TYPE ST_LA_Stellwert :
STRUCT

	Aussenluftklappe_Stellung 		: REAL;
	Bypassklappe_Stellung 			: REAL;
	Register_Ventil_Stellung 		: REAL;
	Sollwert_aktuell 				: REAL;
	Sollwert_berech_aus_Schiebung 	: REAL;
END_STRUCT
END_TYPE

(* stored: Version 1.1.0.1, ProductVersion 3.1.4024.9
   DUT ST_LA_Stellwert: Id {35ade80e-7ae2-4e63-bc1a-fc01a1d80940} *)
